TYPE MachineComSubscribe :
STRUCT
  Request : MachineComRequest; // contains booleans that are used to start a specific sequence.
  Equipment : MachineComSubscribeEquipment;  // structs for equipment objects which are used by the bridges
END_STRUCT
END_TYPE

(* stored: Version 1.1.0.1
   DUT MachineComSubscribe: Id {d547b759-c92d-43bc-b030-f77a6f4e0d30} *)
